FUNCTION_BLOCK FB_Devices
VAR
	devValveV2012 : DEV_Valve := (TagName := 'V2012', Description := 'Standard Valve', TagID := 1);
	devValveV2020 : DEV_Valve := (TagName := 'V2020', Description := 'Standard Valve', TagID := 2);
	devValveV2021 : DEV_Valve := (TagName := 'V2021', Description := 'Standard Valve', TagID := 3);
	devValveV2022 : DEV_Valve := (TagName := 'V2022', Description := 'Standard Valve', TagID := 4);
END_VAR

devValveV2012();
devValveV2020();
devValveV2021();
devValveV2020();

END_FUNCTION_BLOCK

(* stored: Version 1.1.0.1, ProductVersion 3.1.4024.12
   POU FB_Devices: Id {5a1a6b57-ea7a-4b81-b40d-043e4cf8b574}, SpecialFunc None *)
